VAR_GLOBAL
	XAxisEnable:BOOL;
	XAxisJogPos:BOOL;
	XAxisJogNeg:BOOL;
	
END_VAR

(* stored: Version 1.1.0.1, ProductVersion 3.1.4024.2
   GVL GVL_axisContr: Id {ca756a2c-c8a6-46eb-85ff-6e715447bb99} *)
